FUNCTION F_LogL9 
VAR_INPUT
	eLogLevel		: E_LogLevel;
	sLogger			: T_MaxString;
	sMessage		: T_MaxString;
	stArg1			: T_Arg;
	stArg2			: T_Arg;
	stArg3			: T_Arg;
	stArg4			: T_Arg;
	stArg5			: T_Arg;
	stArg6			: T_Arg;
	stArg7			: T_Arg;
	stArg8			: T_Arg;
	stArg9			: T_Arg;
END_VAR

F_LogTArg(
	eLogLevel, 
	sLogger, 
	sMessage, 
	stArg1, 
	stArg2, 
	stArg3, 
	stArg4, 
	stArg5, 
	stArg6, 
	stArg7, 
	stArg8, 
	stArg9, 
	Tc2_Utilities.EMPTY_ARG_VALUE, 
	0
);

END_FUNCTION

(* stored: Version 1.1.0.1, ProductVersion 3.1.4024.6
   POU F_LogL9: Id {fb2f8e79-ae3a-4a1e-8464-9cd32f59a6a1}, SpecialFunc None *)
